PROGRAM MAIN
VAR
	bValue : BOOL;
	{attribute 'pytmc' := 'pv: PLC:TEST:iCount'}
	iCount : INT;
END_VAR

iCount := iCount + 1;

END_PROGRAM

(* stored: Version 1.1.0.1, ProductVersion 3.1.4024.12
   POU MAIN: Id {2f91f540-04e5-4ebb-a672-ddc63ea86f99}, SpecialFunc None *)
